# B&R Automation Studio project DuctLines (part 6)

#### Cyclic.ld
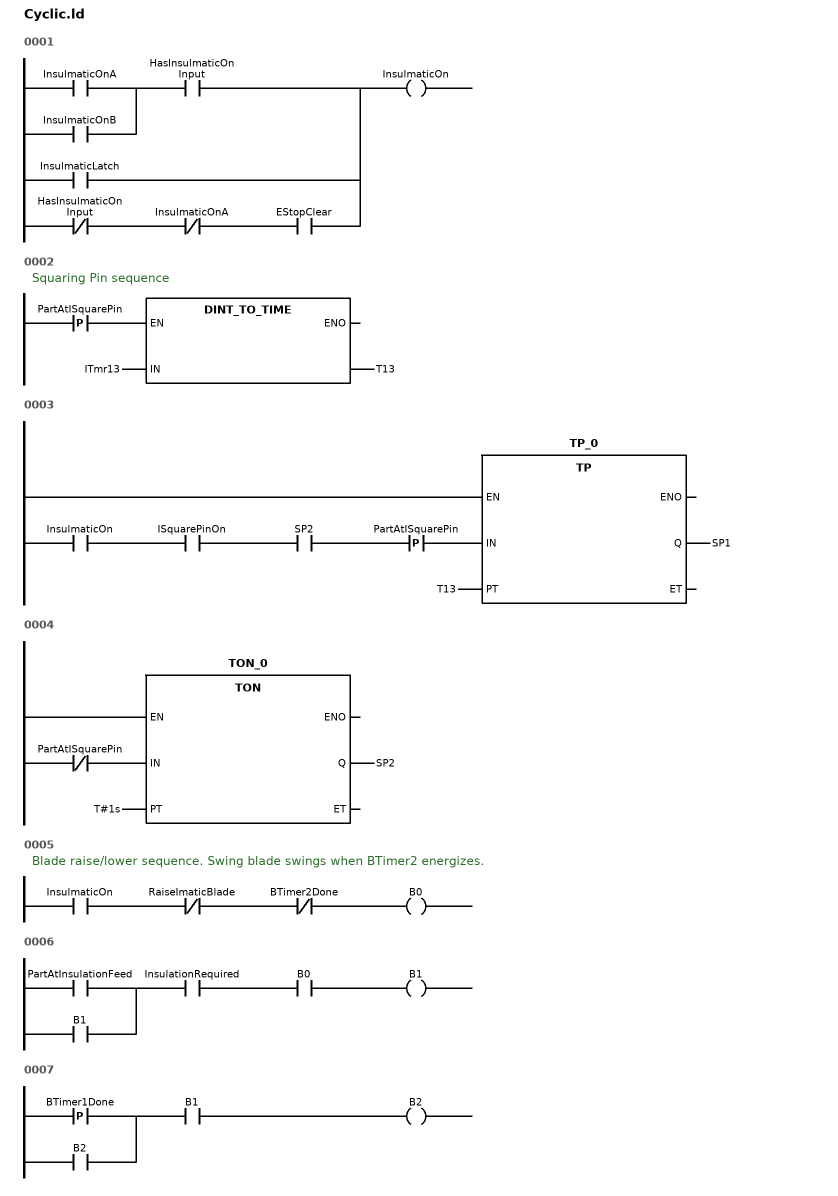
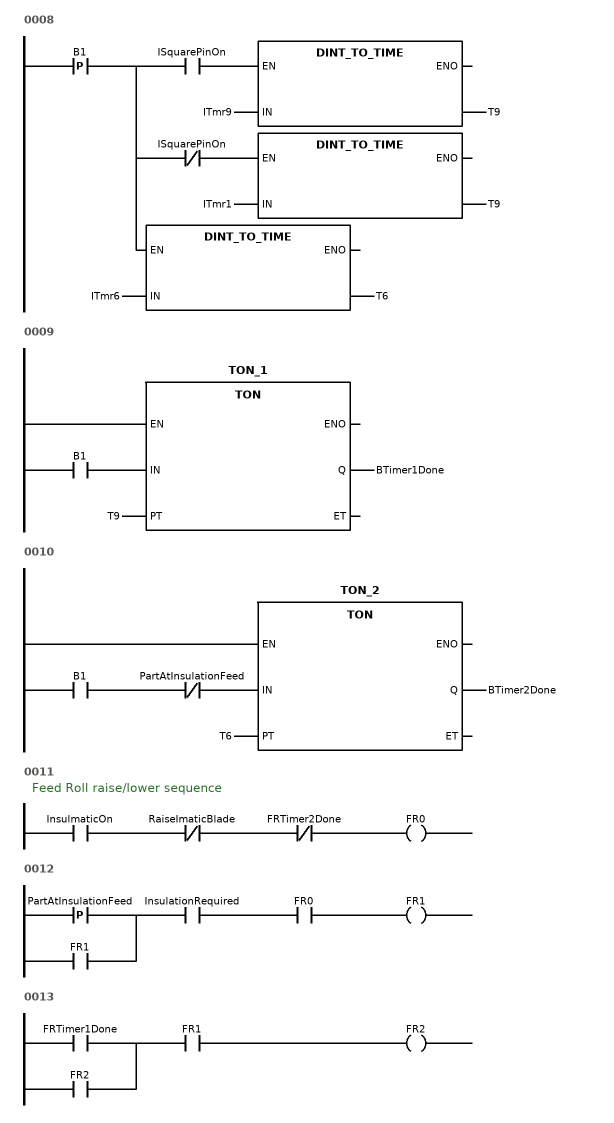
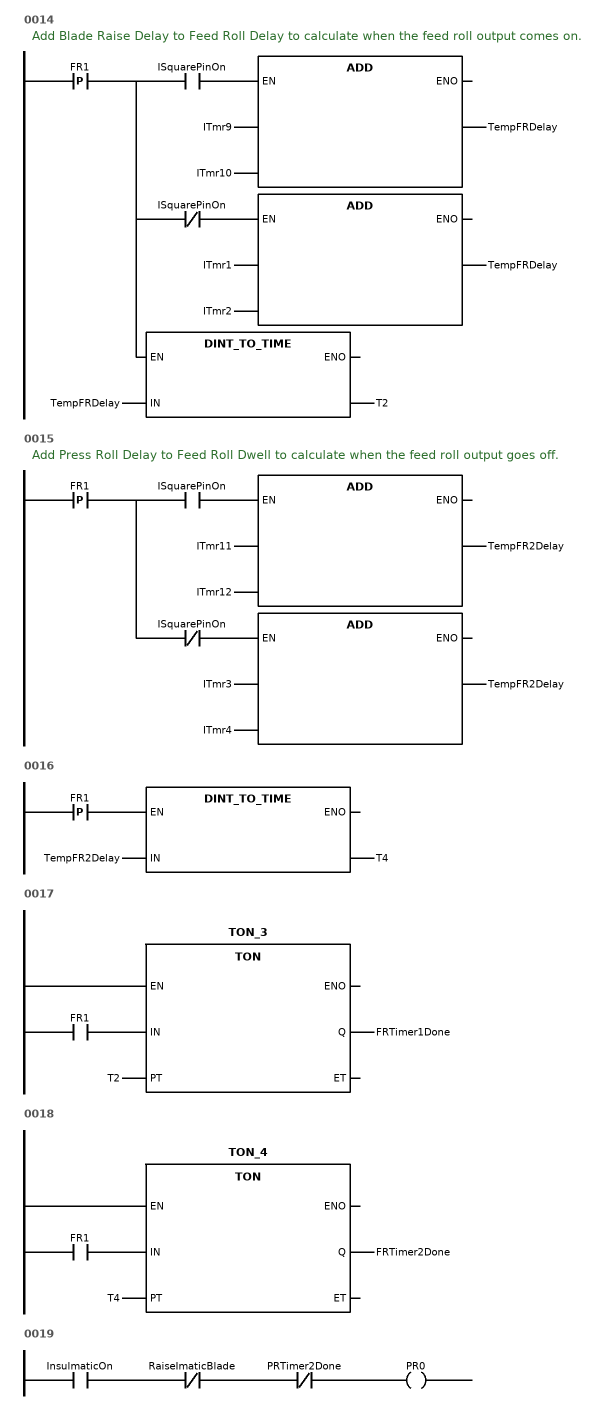
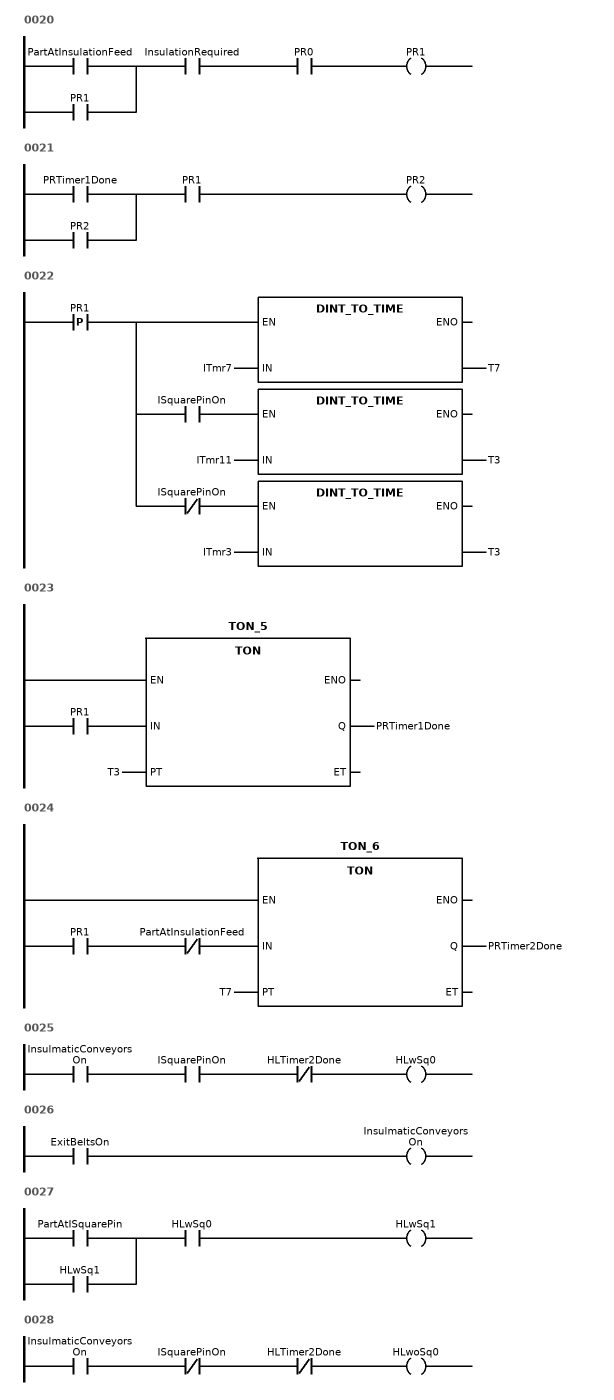
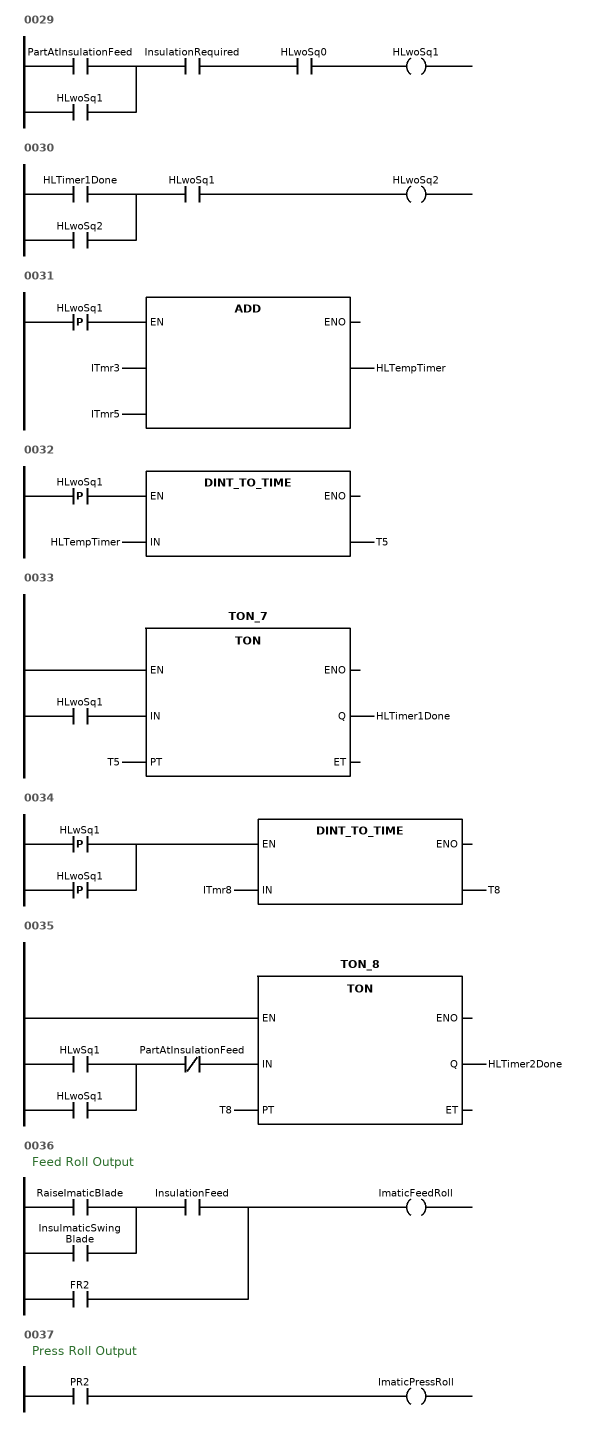
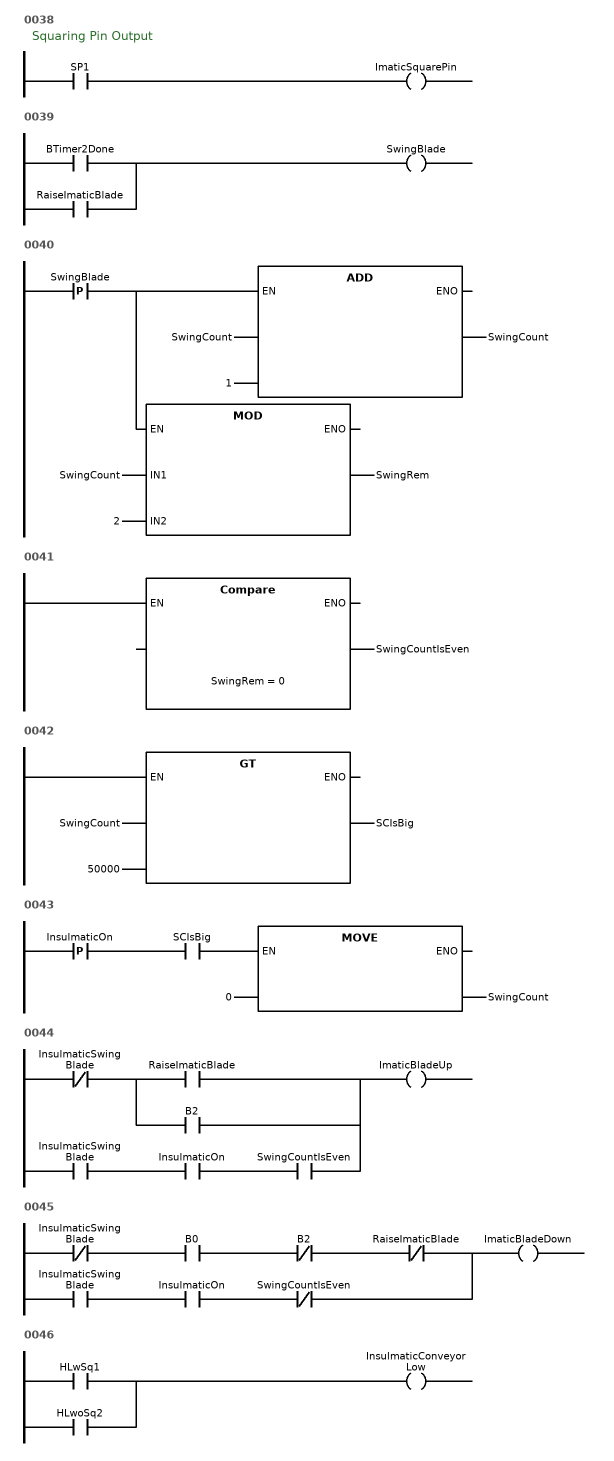
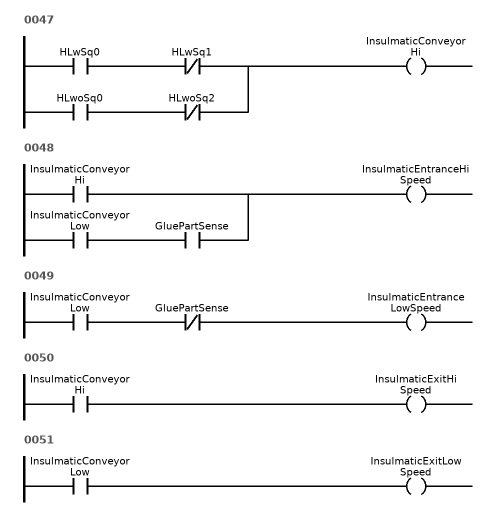
Ladder, written as Structured Text:
```iecst
PROGRAM _CYCLIC
VAR
    _e1 : R_TRIG;
    _e2 : R_TRIG;
    _e3 : R_TRIG;
    _e4 : R_TRIG;
    _e5 : R_TRIG;
    _e6 : R_TRIG;
    _e7 : R_TRIG;
    _e8 : R_TRIG;
    _e9 : R_TRIG;
    _e10 : R_TRIG;
    _e11 : R_TRIG;
    _e12 : R_TRIG;
    _e13 : R_TRIG;
    _e14 : R_TRIG;
    _e15 : R_TRIG;
END_VAR
(* Network 1 *)
InsulmaticOn := ((InsulmaticOnA OR InsulmaticOnB) AND HasInsulmaticOnInput) OR InsulmaticLatch OR (NOT HasInsulmaticOnInput AND NOT InsulmaticOnA AND EStopClear);

(* Network 2: Squaring Pin sequence *)
_e1(CLK := PartAtISquarePin);
IF _e1.Q THEN T13 := DINT_TO_TIME(ITmr13); END_IF;

(* Network 3 *)
_e2(CLK := PartAtISquarePin);
TP_0(IN := InsulmaticOn AND ISquarePinOn AND SP2 AND _e2.Q, PT := T13);
SP1 := TP_0.Q;

(* Network 4 *)
TON_0(IN := NOT PartAtISquarePin, PT := T#1s);
SP2 := TON_0.Q;

(* Network 5: Blade raise/lower sequence. Swing blade swings when BTimer2 energizes. *)
B0 := InsulmaticOn AND NOT RaiseImaticBlade AND NOT BTimer2Done;

(* Network 6 *)
B1 := (PartAtInsulationFeed OR B1) AND InsulationRequired AND B0;

(* Network 7 *)
_e3(CLK := BTimer1Done);
B2 := (_e3.Q OR B2) AND B1;

(* Network 8 *)
_e4(CLK := B1);
IF _e4.Q AND ISquarePinOn THEN T9 := DINT_TO_TIME(ITmr9); END_IF;
IF _e4.Q AND NOT ISquarePinOn THEN T9 := DINT_TO_TIME(ITmr1); END_IF;
IF _e4.Q THEN T6 := DINT_TO_TIME(ITmr6); END_IF;

(* Network 9 *)
TON_1(IN := B1, PT := T9);
BTimer1Done := TON_1.Q;

(* Network 10 *)
TON_2(IN := B1 AND NOT PartAtInsulationFeed, PT := T6);
BTimer2Done := TON_2.Q;

(* Network 11: Feed Roll raise/lower sequence *)
FR0 := InsulmaticOn AND NOT RaiseImaticBlade AND NOT FRTimer2Done;

(* Network 12 *)
_e5(CLK := PartAtInsulationFeed);
FR1 := (_e5.Q OR FR1) AND InsulationRequired AND FR0;

(* Network 13 *)
FR2 := (FRTimer1Done OR FR2) AND FR1;

(* Network 14: Add Blade Raise Delay to Feed Roll Delay to calculate when the feed roll output comes on. *)
_e6(CLK := FR1);
IF _e6.Q AND ISquarePinOn THEN TempFRDelay := ITmr9 + ITmr10; END_IF;
IF _e6.Q AND NOT ISquarePinOn THEN TempFRDelay := ITmr1 + ITmr2; END_IF;
IF _e6.Q THEN T2 := DINT_TO_TIME(TempFRDelay); END_IF;

(* Network 15: Add Press Roll Delay to Feed Roll Dwell to calculate when the feed roll output goes off. *)
_e7(CLK := FR1);
IF _e7.Q AND ISquarePinOn THEN TempFR2Delay := ITmr11 + ITmr12; END_IF;
IF _e7.Q AND NOT ISquarePinOn THEN TempFR2Delay := ITmr3 + ITmr4; END_IF;

(* Network 16 *)
_e8(CLK := FR1);
IF _e8.Q THEN T4 := DINT_TO_TIME(TempFR2Delay); END_IF;

(* Network 17 *)
TON_3(IN := FR1, PT := T2);
FRTimer1Done := TON_3.Q;

(* Network 18 *)
TON_4(IN := FR1, PT := T4);
FRTimer2Done := TON_4.Q;

(* Network 19 *)
PR0 := InsulmaticOn AND NOT RaiseImaticBlade AND NOT PRTimer2Done;

(* Network 20 *)
PR1 := (PartAtInsulationFeed OR PR1) AND InsulationRequired AND PR0;

(* Network 21 *)
PR2 := (PRTimer1Done OR PR2) AND PR1;

(* Network 22 *)
_e9(CLK := PR1);
IF _e9.Q THEN T7 := DINT_TO_TIME(ITmr7); END_IF;
IF _e9.Q AND ISquarePinOn THEN T3 := DINT_TO_TIME(ITmr11); END_IF;
IF _e9.Q AND NOT ISquarePinOn THEN T3 := DINT_TO_TIME(ITmr3); END_IF;

(* Network 23 *)
TON_5(IN := PR1, PT := T3);
PRTimer1Done := TON_5.Q;

(* Network 24 *)
TON_6(IN := PR1 AND NOT PartAtInsulationFeed, PT := T7);
PRTimer2Done := TON_6.Q;

(* Network 25 *)
HLwSq0 := InsulmaticConveyorsOn AND ISquarePinOn AND NOT HLTimer2Done;

(* Network 26 *)
InsulmaticConveyorsOn := ExitBeltsOn;

(* Network 27 *)
HLwSq1 := (PartAtISquarePin OR HLwSq1) AND HLwSq0;

(* Network 28 *)
HLwoSq0 := InsulmaticConveyorsOn AND NOT ISquarePinOn AND NOT HLTimer2Done;

(* Network 29 *)
HLwoSq1 := (PartAtInsulationFeed OR HLwoSq1) AND InsulationRequired AND HLwoSq0;

(* Network 30 *)
HLwoSq2 := (HLTimer1Done OR HLwoSq2) AND HLwoSq1;

(* Network 31 *)
_e10(CLK := HLwoSq1);
IF _e10.Q THEN HLTempTimer := ITmr3 + ITmr5; END_IF;

(* Network 32 *)
_e11(CLK := HLwoSq1);
IF _e11.Q THEN T5 := DINT_TO_TIME(HLTempTimer); END_IF;

(* Network 33 *)
TON_7(IN := HLwoSq1, PT := T5);
HLTimer1Done := TON_7.Q;

(* Network 34 *)
_e12(CLK := HLwSq1);
_e13(CLK := HLwoSq1);
IF _e12.Q OR _e13.Q THEN T8 := DINT_TO_TIME(ITmr8); END_IF;

(* Network 35 *)
TON_8(IN := (HLwSq1 OR HLwoSq1) AND NOT PartAtInsulationFeed, PT := T8);
HLTimer2Done := TON_8.Q;

(* Network 36: Feed Roll Output *)
ImaticFeedRoll := ((RaiseImaticBlade OR InsulmaticSwingBlade) AND InsulationFeed) OR FR2;

(* Network 37: Press Roll Output *)
ImaticPressRoll := PR2;

(* Network 38: Squaring Pin Output *)
ImaticSquarePin := SP1;

(* Network 39 *)
SwingBlade := BTimer2Done OR RaiseImaticBlade;

(* Network 40 *)
_e14(CLK := SwingBlade);
IF _e14.Q THEN
    SwingCount := SwingCount + 1;
    SwingRem := SwingCount MOD 2;
END_IF;

(* Network 41 *)
SwingCountIsEven := SwingRem = 0;

(* Network 42 *)
SCIsBig := SwingCount > 50000;

(* Network 43 *)
_e15(CLK := InsulmaticOn);
IF _e15.Q AND SCIsBig THEN SwingCount := 0; END_IF;

(* Network 44 *)
ImaticBladeUp := (NOT InsulmaticSwingBlade AND (RaiseImaticBlade OR B2)) OR (InsulmaticSwingBlade AND InsulmaticOn AND SwingCountIsEven);

(* Network 45 *)
ImaticBladeDown := (NOT InsulmaticSwingBlade AND B0 AND NOT B2 AND NOT RaiseImaticBlade) OR (InsulmaticSwingBlade AND InsulmaticOn AND NOT SwingCountIsEven);

(* Network 46 *)
InsulmaticConveyorLow := HLwSq1 OR HLwoSq2;

(* Network 47 *)
InsulmaticConveyorHi := (HLwSq0 AND NOT HLwSq1) OR (HLwoSq0 AND NOT HLwoSq2);

(* Network 48 *)
InsulmaticEntranceHiSpeed := InsulmaticConveyorHi OR (InsulmaticConveyorLow AND GluePartSense);

(* Network 49 *)
InsulmaticEntranceLowSpeed := InsulmaticConveyorLow AND NOT GluePartSense;

(* Network 50 *)
InsulmaticExitHiSpeed := InsulmaticConveyorHi;

(* Network 51 *)
InsulmaticExitLowSpeed := InsulmaticConveyorLow;
END_PROGRAM
```

### Program Logical/Pinspotter (IEC)

#### Variables.var
```iecst
VAR
	PS0 : BOOL;
	EncoderReset : BOOL;
	PS1 : BOOL;
	PinSpaceSelector : USINT;
	RepeatCounter : DINT;
	Target : DINT;
	PinSpacing : REAL;
	PinSpaceSelectorIs9 : BOOL;
	RealTarget : REAL;
	RealCounts : REAL;
	Drive : BOOL;
	DriveComplete : BOOL;
	DriveDwell : TIME;
	PS3 : BOOL;
	PS2 : BOOL;
	UpDateSignal : BOOL;
	IndexFinished : BOOL;
	PinningDone : BOOL;
	PS4 : BOOL;
	PinAgain : BOOL;
	TON_2 : TON;
	DelayTime : TIME;
	TP_1 : TP;
	LoadDelayPulse : BOOL;
	PinLoadTime : TIME;
	TP_2 : TP;
	TON_0 : TON;
	RCounterIs0 : BOOL;
END_VAR
```

#### Cyclic.ld
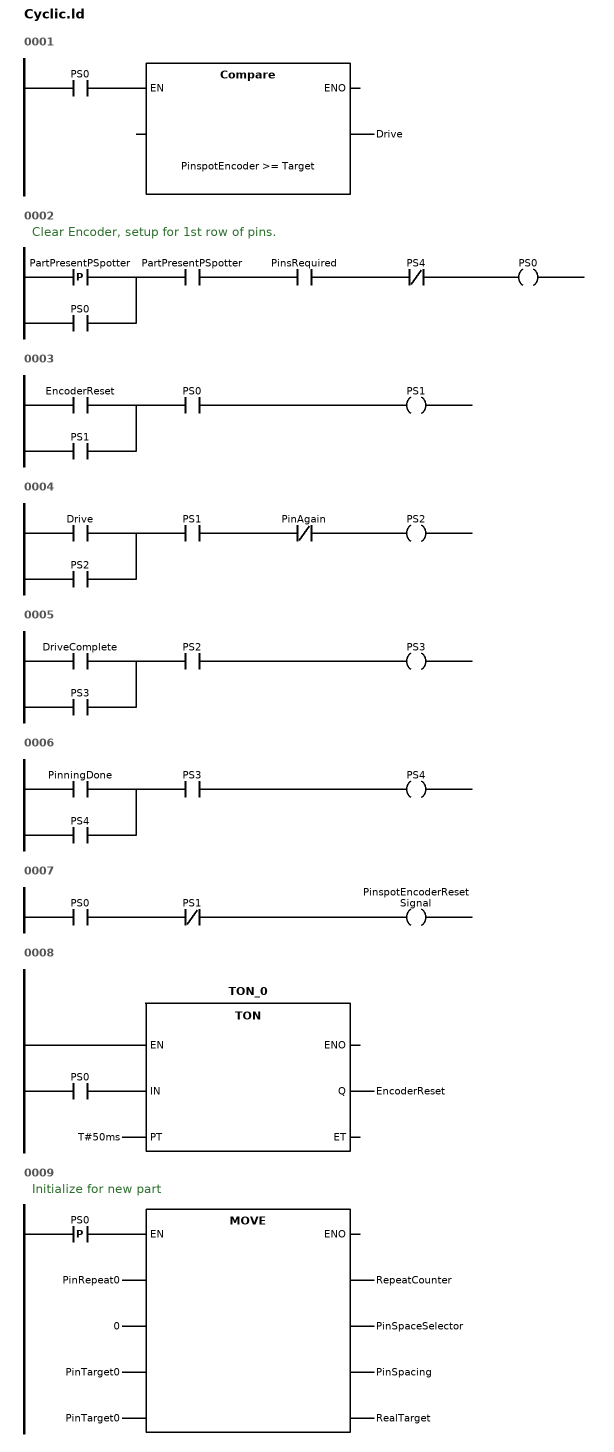
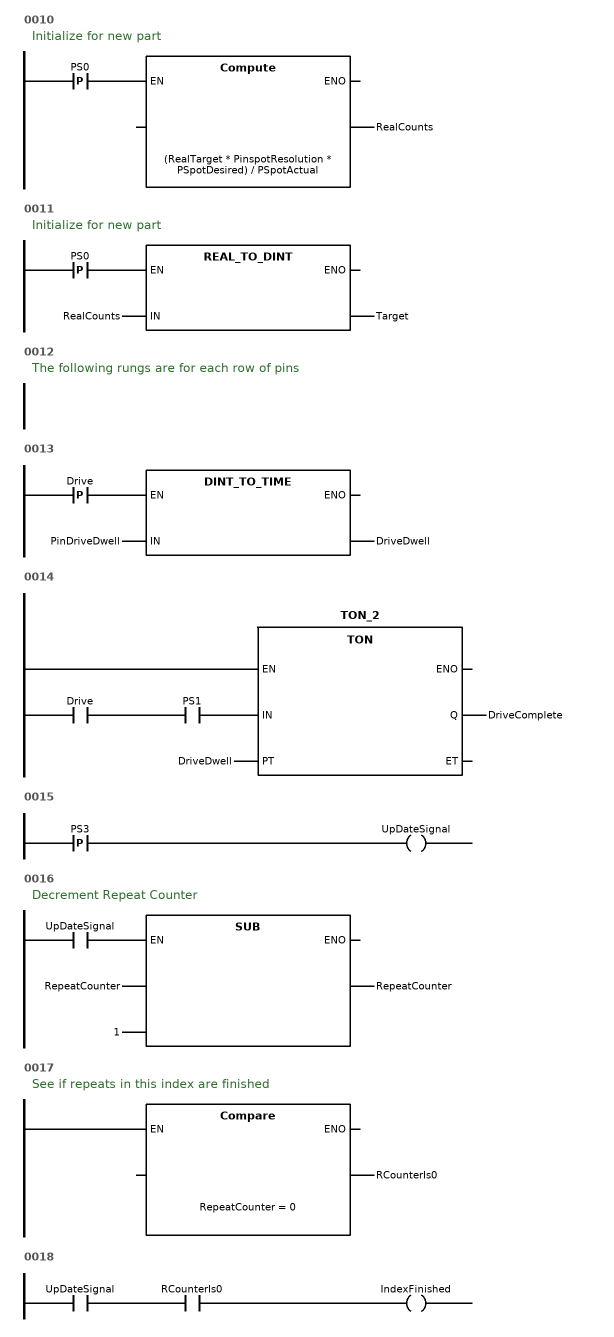
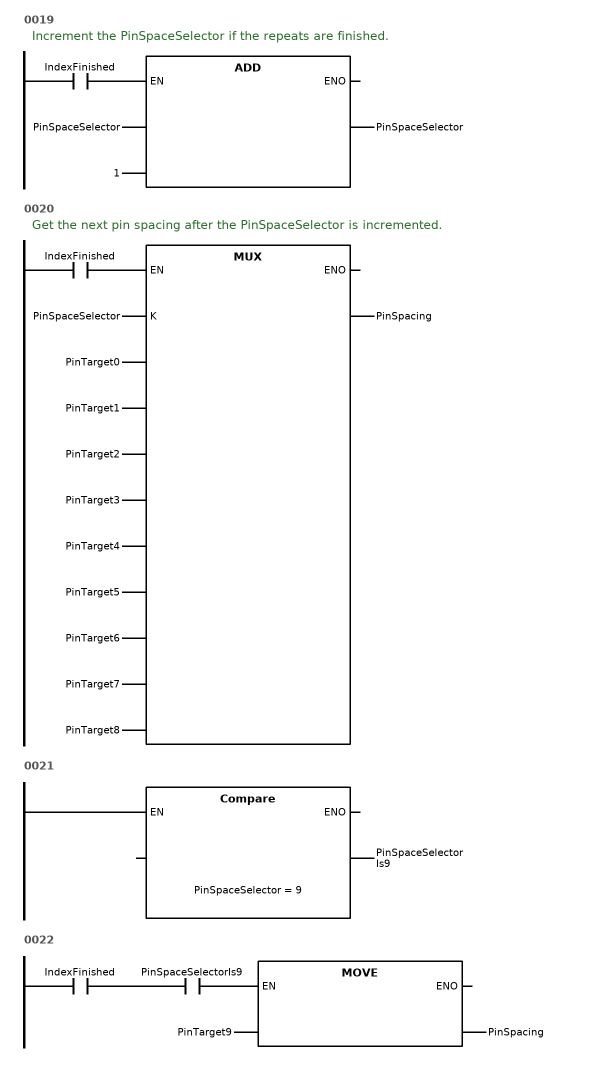
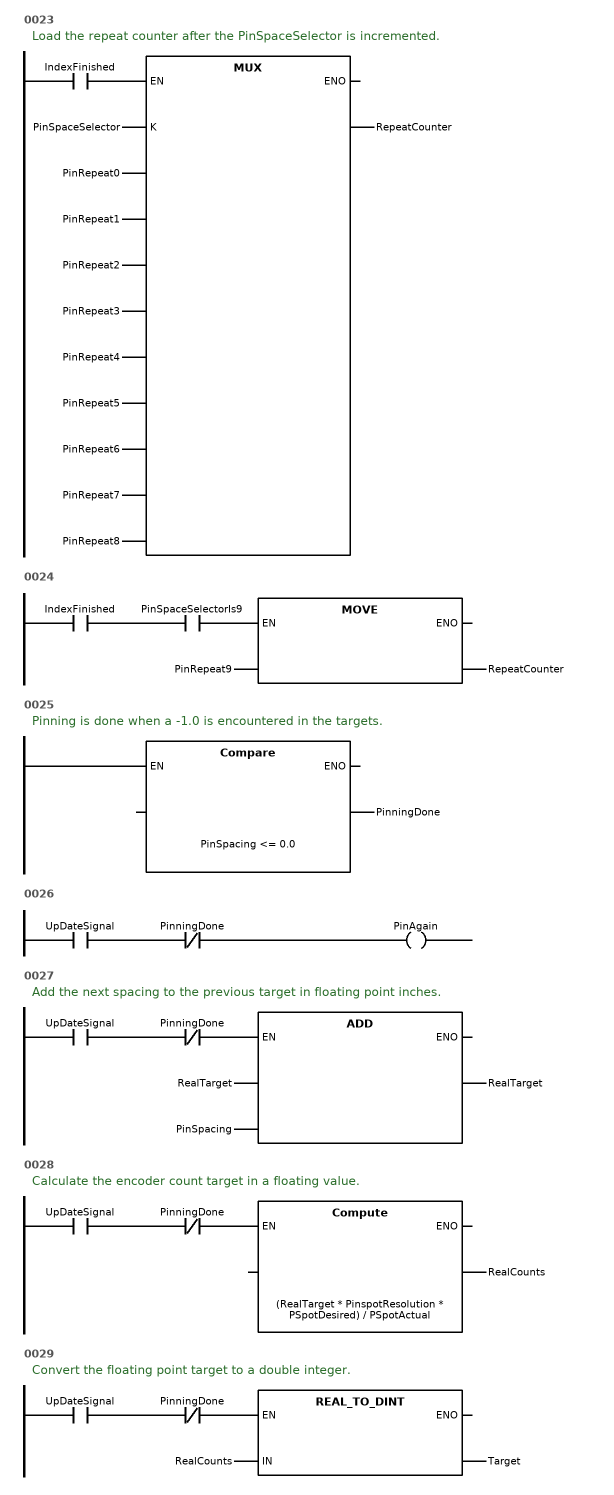
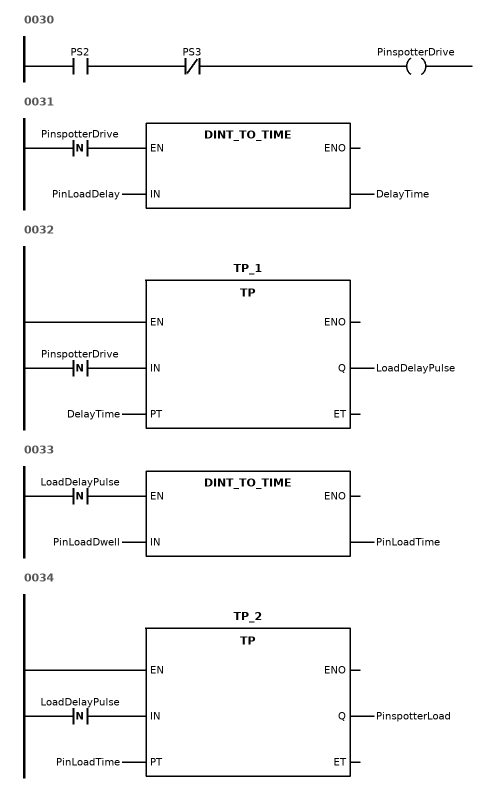
Ladder, written as Structured Text:
```iecst
PROGRAM _CYCLIC
VAR
    _e1 : R_TRIG;
    _e2 : R_TRIG;
    _e3 : R_TRIG;
    _e4 : R_TRIG;
    _e5 : R_TRIG;
    _e6 : R_TRIG;
    _e7 : F_TRIG;
    _e8 : F_TRIG;
    _e9 : F_TRIG;
    _e10 : F_TRIG;
END_VAR
(* Network 1 *)
IF PS0 THEN Drive := PinspotEncoder >= Target; END_IF;

(* Network 2: Clear Encoder, setup for 1st row of pins. *)
_e1(CLK := PartPresentPSpotter);
PS0 := (_e1.Q OR PS0) AND PartPresentPSpotter AND PinsRequired AND NOT PS4;

(* Network 3 *)
PS1 := (EncoderReset OR PS1) AND PS0;

(* Network 4 *)
PS2 := (Drive OR PS2) AND PS1 AND NOT PinAgain;

(* Network 5 *)
PS3 := (DriveComplete OR PS3) AND PS2;

(* Network 6 *)
PS4 := (PinningDone OR PS4) AND PS3;

(* Network 7 *)
PinspotEncoderResetSignal := PS0 AND NOT PS1;

(* Network 8 *)
TON_0(IN := PS0, PT := T#50ms);
EncoderReset := TON_0.Q;

(* Network 9: Initialize for new part *)
_e2(CLK := PS0);
IF _e2.Q THEN
    RepeatCounter := PinRepeat0;
    PinSpaceSelector := 0;
    PinSpacing := PinTarget0;
    RealTarget := PinTarget0;
END_IF;

(* Network 10: Initialize for new part *)
_e3(CLK := PS0);
IF _e3.Q THEN RealCounts := (RealTarget * PinspotResolution * PSpotDesired) / PSpotActual; END_IF;

(* Network 11: Initialize for new part *)
_e4(CLK := PS0);
IF _e4.Q THEN Target := REAL_TO_DINT(RealCounts); END_IF;

(* Network 12: The following rungs are for each row of pins *)

(* Network 13 *)
_e5(CLK := Drive);
IF _e5.Q THEN DriveDwell := DINT_TO_TIME(PinDriveDwell); END_IF;

(* Network 14 *)
TON_2(IN := Drive AND PS1, PT := DriveDwell);
DriveComplete := TON_2.Q;

(* Network 15 *)
_e6(CLK := PS3);
UpDateSignal := _e6.Q;

(* Network 16: Decrement Repeat Counter *)
IF UpDateSignal THEN RepeatCounter := RepeatCounter - 1; END_IF;

(* Network 17: See if repeats in this index are finished *)
RCounterIs0 := RepeatCounter = 0;

(* Network 18 *)
IndexFinished := UpDateSignal AND RCounterIs0;

(* Network 19: Increment the PinSpaceSelector if the repeats are finished. *)
IF IndexFinished THEN PinSpaceSelector := PinSpaceSelector + 1; END_IF;

(* Network 20: Get the next pin spacing after the PinSpaceSelector is incremented. *)
IF IndexFinished THEN
    PinSpacing := MUX(K := PinSpaceSelector, IN2 := PinTarget0, IN3 := PinTarget1, IN4 := PinTarget2, IN5 := PinTarget3, IN6 := PinTarget4, IN7 := PinTarget5, IN8 := PinTarget6, IN9 := PinTarget7, IN10 := PinTarget8);
END_IF;

(* Network 21 *)
PinSpaceSelectorIs9 := PinSpaceSelector = 9;

(* Network 22 *)
IF IndexFinished AND PinSpaceSelectorIs9 THEN PinSpacing := PinTarget9; END_IF;

(* Network 23: Load the repeat counter after the PinSpaceSelector is incremented. *)
IF IndexFinished THEN
    RepeatCounter := MUX(K := PinSpaceSelector, IN2 := PinRepeat0, IN3 := PinRepeat1, IN4 := PinRepeat2, IN5 := PinRepeat3, IN6 := PinRepeat4, IN7 := PinRepeat5, IN8 := PinRepeat6, IN9 := PinRepeat7, IN10 := PinRepeat8);
END_IF;

(* Network 24 *)
IF IndexFinished AND PinSpaceSelectorIs9 THEN RepeatCounter := PinRepeat9; END_IF;

(* Network 25: Pinning is done when a -1.0 is encountered in the targets. *)
PinningDone := PinSpacing <= 0.0;

(* Network 26 *)
PinAgain := UpDateSignal AND NOT PinningDone;

(* Network 27: Add the next spacing to the previous target in floating point inches. *)
IF UpDateSignal AND NOT PinningDone THEN RealTarget := RealTarget + PinSpacing; END_IF;

(* Network 28: Calculate the encoder count target in a floating value.  *)
IF UpDateSignal AND NOT PinningDone THEN
    RealCounts := (RealTarget * PinspotResolution * PSpotDesired) / PSpotActual;
END_IF;

(* Network 29: Convert the floating point target to a double integer. *)
IF UpDateSignal AND NOT PinningDone THEN Target := REAL_TO_DINT(RealCounts); END_IF;

(* Network 30 *)
PinspotterDrive := PS2 AND NOT PS3;

(* Network 31 *)
_e7(CLK := PinspotterDrive);
IF _e7.Q THEN DelayTime := DINT_TO_TIME(PinLoadDelay); END_IF;

(* Network 32 *)
_e8(CLK := PinspotterDrive);
TP_1(IN := _e8.Q, PT := DelayTime);
LoadDelayPulse := TP_1.Q;

(* Network 33 *)
_e9(CLK := LoadDelayPulse);
IF _e9.Q THEN PinLoadTime := DINT_TO_TIME(PinLoadDwell); END_IF;

(* Network 34 *)
_e10(CLK := LoadDelayPulse);
TP_2(IN := _e10.Q, PT := PinLoadTime);
PinspotterLoad := TP_2.Q;
END_PROGRAM
```

### Program Logical/BrakeCommon (IEC) - In this file: The encoder feedback is scaled to inches. All of the brakes use real dimensions, except for the Electric Servo Brake, The Auto Latch for all brake styles, Target selection for all brake styles, A latch that holds all outputs in their initial state, The bending routine for all brakes without their own PLC begins about rung 29, Clamp, Leaf, Beam outputs for brakes without a PLC begins about rung 42, Brake Conveyor and Auto/Man Indicator Outputs

#### Variables.var
```iecst
VAR
	BAOK : BOOL;
	BCTGreatThan0 : BOOL;
	BDOK : BOOL;
	BeamSettleTimerDone : BOOL;
	BrakeSetOK : BOOL;
	EWBAutoLatch : BOOL;
	JobsDifferent : BOOL;
	MakeTargets : BOOL;
	RaiseLeafTimerDone : BOOL;
	RawBrakeEncoder : REAL;
	RefSignalReset : BOOL;
	ResOK : BOOL;
	SetSignalReset : BOOL;
	SingleCyclingBrake : BOOL;
	StopLeafTimerDone : BOOL;
	TON_0 : TON;
	TON_1 : TON;
	TON_2 : TON;
	TON_3 : TON;
	TON_4 : TON;
	WBBeamSettleStep : BOOL;
	WBCheckBeamStep : BOOL;
	WBCheckLeafStep : BOOL;
	WBIndex : INT;
	WBLeafNotHomeStep : BOOL;
	WBLowerBeamStep : BOOL;
	WBLowerLeafStep : BOOL;
	WBRaiseBeamStep : BOOL;
	WBStopLeafStep : BOOL;
END_VAR
```

#### Cyclic.ld
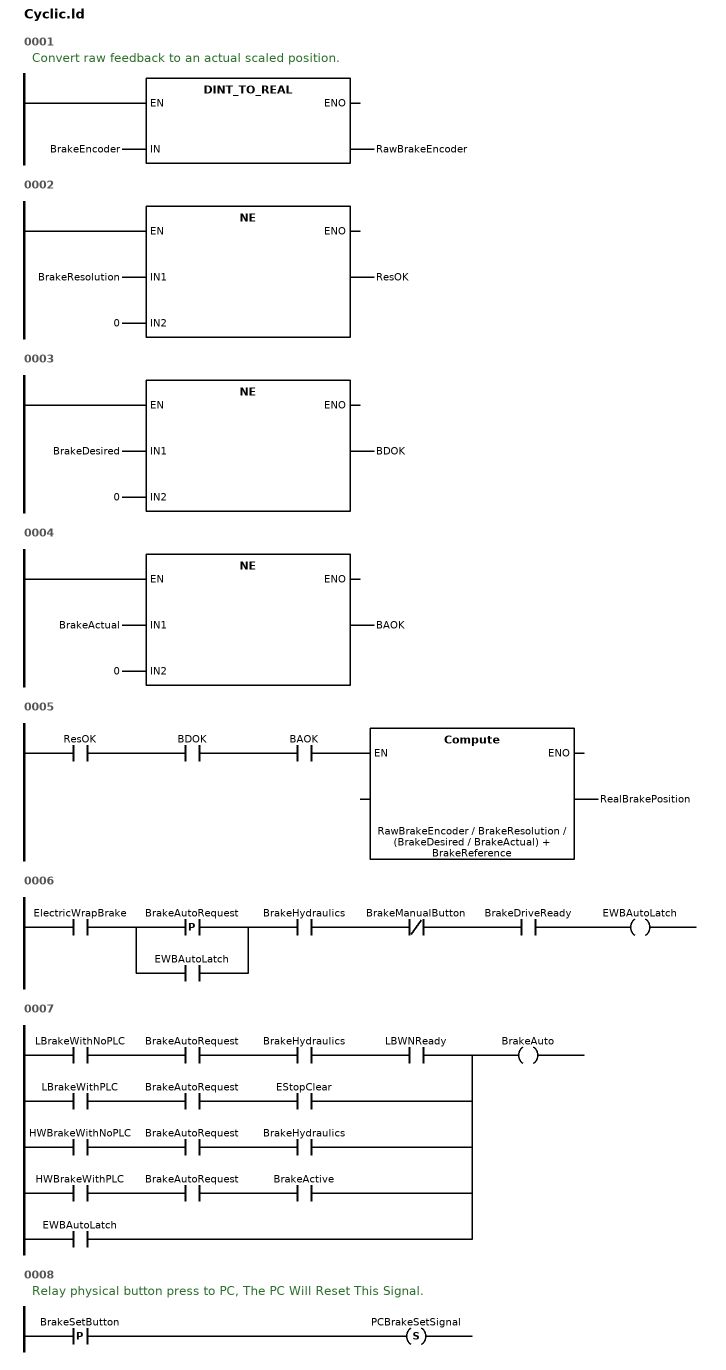
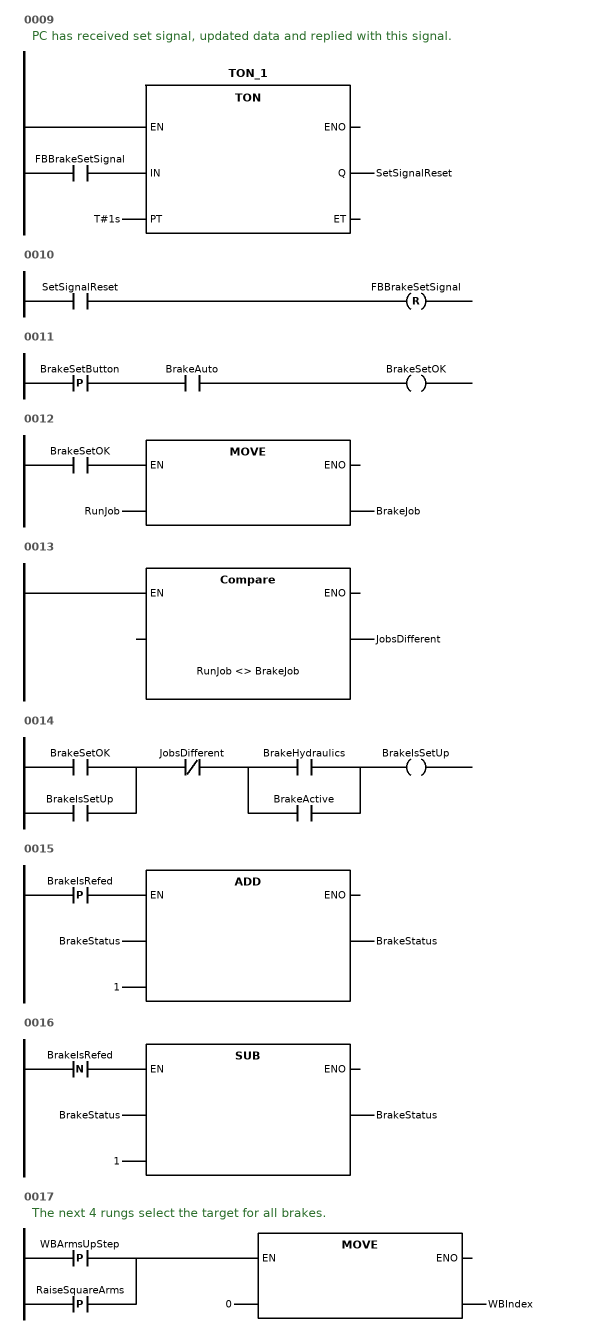
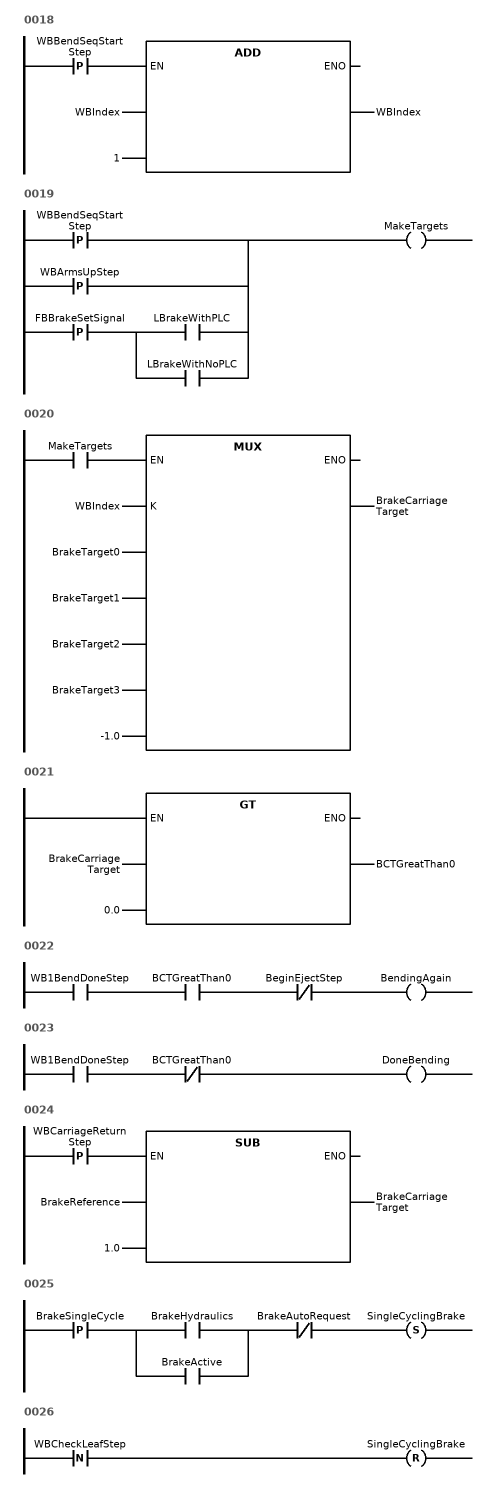
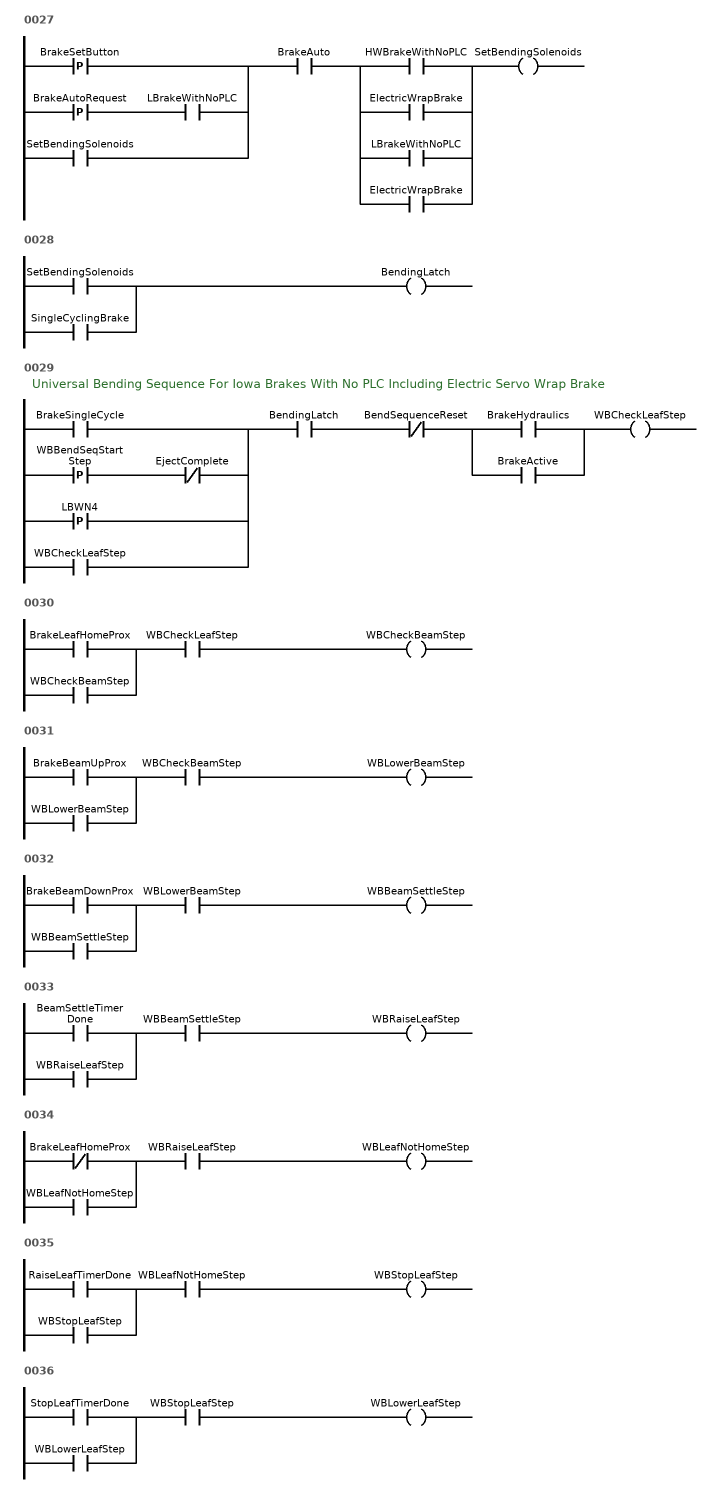
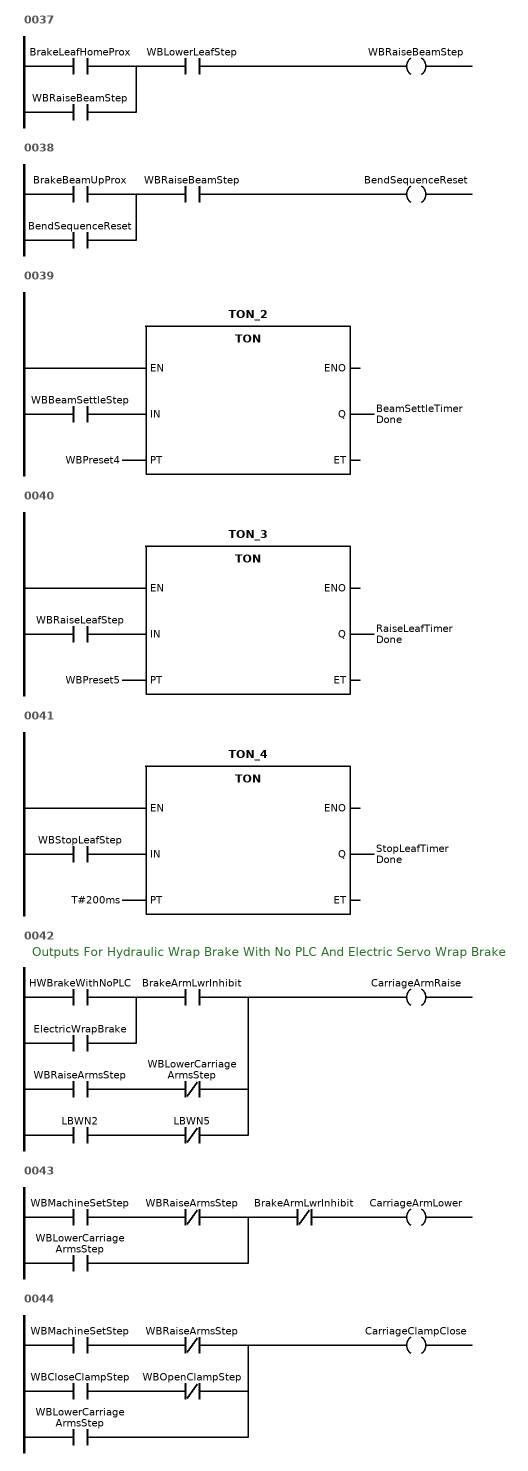
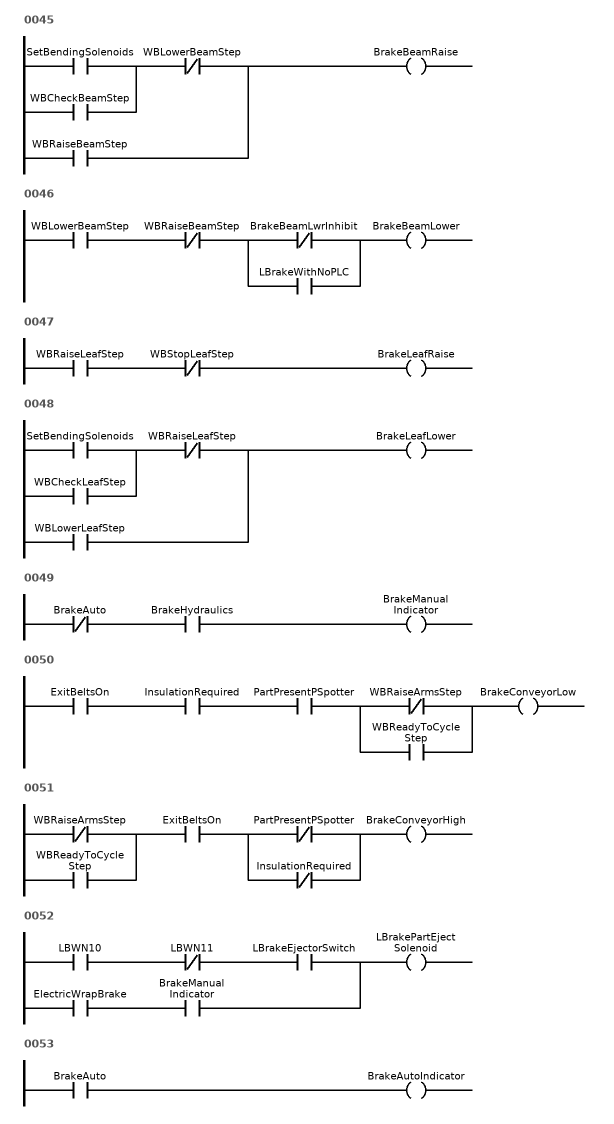
Ladder, written as Structured Text:
```iecst
PROGRAM _CYCLIC
VAR
    _e1 : R_TRIG;
    _e2 : R_TRIG;
    _e3 : R_TRIG;
    _p4 : BOOL;
    _e5 : R_TRIG;
    _e6 : F_TRIG;
    _e7 : R_TRIG;
    _e8 : R_TRIG;
    _e9 : R_TRIG;
    _e10 : R_TRIG;
    _e11 : R_TRIG;
    _e12 : R_TRIG;
    _e13 : R_TRIG;
    _e14 : R_TRIG;
    _e15 : F_TRIG;
    _e16 : R_TRIG;
    _e17 : R_TRIG;
    _p18 : BOOL;
    _e19 : R_TRIG;
    _e20 : R_TRIG;
    _p21 : BOOL;
    _p22 : BOOL;
    _p23 : BOOL;
END_VAR
(* Network 1: Convert raw feedback to an actual scaled position. *)
RawBrakeEncoder := DINT_TO_REAL(BrakeEncoder);

(* Network 2 *)
ResOK := BrakeResolution <> 0;

(* Network 3 *)
BDOK := BrakeDesired <> 0;

(* Network 4 *)
BAOK := BrakeActual <> 0;

(* Network 5 *)
IF ResOK AND BDOK AND BAOK THEN
    RealBrakePosition := RawBrakeEncoder / BrakeResolution / (BrakeDesired / BrakeActual) + BrakeReference;
END_IF;

(* Network 6 *)
_e1(CLK := BrakeAutoRequest);
EWBAutoLatch := ElectricWrapBrake AND (_e1.Q OR EWBAutoLatch) AND BrakeHydraulics AND NOT BrakeManualButton AND BrakeDriveReady;

(* Network 7 *)
BrakeAuto := (LBrakeWithNoPLC AND BrakeAutoRequest AND BrakeHydraulics AND LBWNReady) OR (LBrakeWithPLC AND BrakeAutoRequest AND EStopClear) OR (HWBrakeWithNoPLC AND BrakeAutoRequest AND BrakeHydraulics) OR (HWBrakeWithPLC AND BrakeAutoRequest AND BrakeActive) OR EWBAutoLatch;

(* Network 8: Relay physical button press to PC, The PC Will Reset This Signal. *)
_e2(CLK := BrakeSetButton);
IF _e2.Q THEN PCBrakeSetSignal := TRUE; END_IF;

(* Network 9: PC has received set signal, updated data and replied with this signal. *)
TON_1(IN := FBBrakeSetSignal, PT := T#1s);
SetSignalReset := TON_1.Q;

(* Network 10 *)
IF SetSignalReset THEN FBBrakeSetSignal := FALSE; END_IF;

(* Network 11 *)
_e3(CLK := BrakeSetButton);
BrakeSetOK := _e3.Q AND BrakeAuto;

(* Network 12 *)
IF BrakeSetOK THEN BrakeJob := RunJob; END_IF;

(* Network 13 *)
JobsDifferent := RunJob <> BrakeJob;

(* Network 14 *)
_p4 := (BrakeSetOK OR BrakeIsSetUp) AND NOT JobsDifferent;
BrakeIsSetUp := _p4 AND (BrakeHydraulics OR BrakeActive);

(* Network 15 *)
_e5(CLK := BrakeIsRefed);
IF _e5.Q THEN BrakeStatus := BrakeStatus + 1; END_IF;

(* Network 16 *)
_e6(CLK := BrakeIsRefed);
IF _e6.Q THEN BrakeStatus := BrakeStatus - 1; END_IF;

(* Network 17: The next 4 rungs select the target for all brakes. *)
_e7(CLK := WBArmsUpStep);
_e8(CLK := RaiseSquareArms);
IF _e7.Q OR _e8.Q THEN WBIndex := 0; END_IF;

(* Network 18 *)
_e9(CLK := WBBendSeqStartStep);
IF _e9.Q THEN WBIndex := WBIndex + 1; END_IF;

(* Network 19 *)
_e10(CLK := WBBendSeqStartStep);
_e11(CLK := WBArmsUpStep);
_e12(CLK := FBBrakeSetSignal);
MakeTargets := _e10.Q OR _e11.Q OR (_e12.Q AND (LBrakeWithPLC OR LBrakeWithNoPLC));

(* Network 20 *)
IF MakeTargets THEN
    BrakeCarriageTarget := MUX(K := WBIndex, IN2 := BrakeTarget0, IN3 := BrakeTarget1, IN4 := BrakeTarget2, IN5 := BrakeTarget3, IN6 := -1.0);
END_IF;

(* Network 21 *)
BCTGreatThan0 := BrakeCarriageTarget > 0.0;

(* Network 22 *)
BendingAgain := WB1BendDoneStep AND BCTGreatThan0 AND NOT BeginEjectStep;

(* Network 23 *)
DoneBending := WB1BendDoneStep AND NOT BCTGreatThan0;

(* Network 24 *)
_e13(CLK := WBCarriageReturnStep);
IF _e13.Q THEN BrakeCarriageTarget := BrakeReference - 1.0; END_IF;

(* Network 25 *)
_e14(CLK := BrakeSingleCycle);
IF _e14.Q AND (BrakeHydraulics OR BrakeActive) AND NOT BrakeAutoRequest THEN
    SingleCyclingBrake := TRUE;
END_IF;

(* Network 26 *)
_e15(CLK := WBCheckLeafStep);
IF _e15.Q THEN SingleCyclingBrake := FALSE; END_IF;

(* Network 27 *)
_e16(CLK := BrakeSetButton);
_e17(CLK := BrakeAutoRequest);
_p18 := (_e16.Q OR (_e17.Q AND LBrakeWithNoPLC) OR SetBendingSolenoids) AND BrakeAuto;
SetBendingSolenoids := _p18 AND (HWBrakeWithNoPLC OR ElectricWrapBrake OR LBrakeWithNoPLC);

(* Network 28 *)
BendingLatch := SetBendingSolenoids OR SingleCyclingBrake;

(* Network 29: Universal Bending Sequence For Iowa Brakes With No PLC Including Electric Servo Wrap Brake *)
_e19(CLK := WBBendSeqStartStep);
_e20(CLK := LBWN4);
_p21 := (BrakeSingleCycle OR (_e19.Q AND NOT EjectComplete) OR _e20.Q OR WBCheckLeafStep) AND BendingLatch AND NOT BendSequenceReset;
WBCheckLeafStep := _p21 AND (BrakeHydraulics OR BrakeActive);

(* Network 30 *)
WBCheckBeamStep := (BrakeLeafHomeProx OR WBCheckBeamStep) AND WBCheckLeafStep;

(* Network 31 *)
WBLowerBeamStep := (BrakeBeamUpProx OR WBLowerBeamStep) AND WBCheckBeamStep;

(* Network 32 *)
WBBeamSettleStep := (BrakeBeamDownProx OR WBBeamSettleStep) AND WBLowerBeamStep;

(* Network 33 *)
WBRaiseLeafStep := (BeamSettleTimerDone OR WBRaiseLeafStep) AND WBBeamSettleStep;

(* Network 34 *)
WBLeafNotHomeStep := (NOT BrakeLeafHomeProx OR WBLeafNotHomeStep) AND WBRaiseLeafStep;

(* Network 35 *)
WBStopLeafStep := (RaiseLeafTimerDone OR WBStopLeafStep) AND WBLeafNotHomeStep;

(* Network 36 *)
WBLowerLeafStep := (StopLeafTimerDone OR WBLowerLeafStep) AND WBStopLeafStep;

(* Network 37 *)
WBRaiseBeamStep := (BrakeLeafHomeProx OR WBRaiseBeamStep) AND WBLowerLeafStep;

(* Network 38 *)
BendSequenceReset := (BrakeBeamUpProx OR BendSequenceReset) AND WBRaiseBeamStep;

(* Network 39 *)
TON_2(IN := WBBeamSettleStep, PT := WBPreset4);
BeamSettleTimerDone := TON_2.Q;

(* Network 40 *)
TON_3(IN := WBRaiseLeafStep, PT := WBPreset5);
RaiseLeafTimerDone := TON_3.Q;

(* Network 41 *)
TON_4(IN := WBStopLeafStep, PT := T#200ms);
StopLeafTimerDone := TON_4.Q;

(* Network 42: Outputs For Hydraulic Wrap Brake With No PLC And Electric Servo Wrap Brake *)
CarriageArmRaise := ((HWBrakeWithNoPLC OR ElectricWrapBrake) AND BrakeArmLwrInhibit) OR (WBRaiseArmsStep AND NOT WBLowerCarriageArmsStep) OR (LBWN2 AND NOT LBWN5);

(* Network 43 *)
CarriageArmLower := ((WBMachineSetStep AND NOT WBRaiseArmsStep) OR WBLowerCarriageArmsStep) AND NOT BrakeArmLwrInhibit;

(* Network 44 *)
CarriageClampClose := (WBMachineSetStep AND NOT WBRaiseArmsStep) OR (WBCloseClampStep AND NOT WBOpenClampStep) OR WBLowerCarriageArmsStep;

(* Network 45 *)
BrakeBeamRaise := ((SetBendingSolenoids OR WBCheckBeamStep) AND NOT WBLowerBeamStep) OR WBRaiseBeamStep;

(* Network 46 *)
BrakeBeamLower := WBLowerBeamStep AND NOT WBRaiseBeamStep AND (NOT BrakeBeamLwrInhibit OR LBrakeWithNoPLC);

(* Network 47 *)
BrakeLeafRaise := WBRaiseLeafStep AND NOT WBStopLeafStep;

(* Network 48 *)
BrakeLeafLower := ((SetBendingSolenoids OR WBCheckLeafStep) AND NOT WBRaiseLeafStep) OR WBLowerLeafStep;

(* Network 49 *)
BrakeManualIndicator := NOT BrakeAuto AND BrakeHydraulics;

(* Network 50 *)
_p22 := ExitBeltsOn AND InsulationRequired AND PartPresentPSpotter;
BrakeConveyorLow := _p22 AND (NOT WBRaiseArmsStep OR WBReadyToCycleStep);

(* Network 51 *)
_p23 := (NOT WBRaiseArmsStep OR WBReadyToCycleStep) AND ExitBeltsOn;
BrakeConveyorHigh := _p23 AND (NOT PartPresentPSpotter OR NOT InsulationRequired);

(* Network 52 *)
LBrakePartEjectSolenoid := (LBWN10 AND NOT LBWN11 AND LBrakeEjectorSwitch) OR (ElectricWrapBrake AND BrakeManualIndicator);

(* Network 53 *)
BrakeAutoIndicator := BrakeAuto;
END_PROGRAM
```

### Program Logical/HWBwoPLC (IEC)

#### Variables.var
```iecst
VAR
	EjectTimerDone : BOOL;
	PositionGreaterThan12 : BOOL;
	PPDTimerDone : BOOL;
	SquareTimerDone : BOOL;
	StartBeltTimerDone : BOOL;
	TON_0 : TON;
	TON_1 : TON;
	TON_2 : TON;
	TON_3 : TON;
	TrailDelay1Done : BOOL;
	TON_4 : TON;
	LBPartSquared : BOOL;
	TON_5 : TON;
	LBBeamDownDone : BOOL;
	TON_6 : TON;
	EjectDwellDone : BOOL;
	LBWN12 : BOOL;
	MoveStarted : BOOL;
	TON_7 : TON;
	ReturnMoveStart : BOOL;
END_VAR
```

#### Cyclic.ld
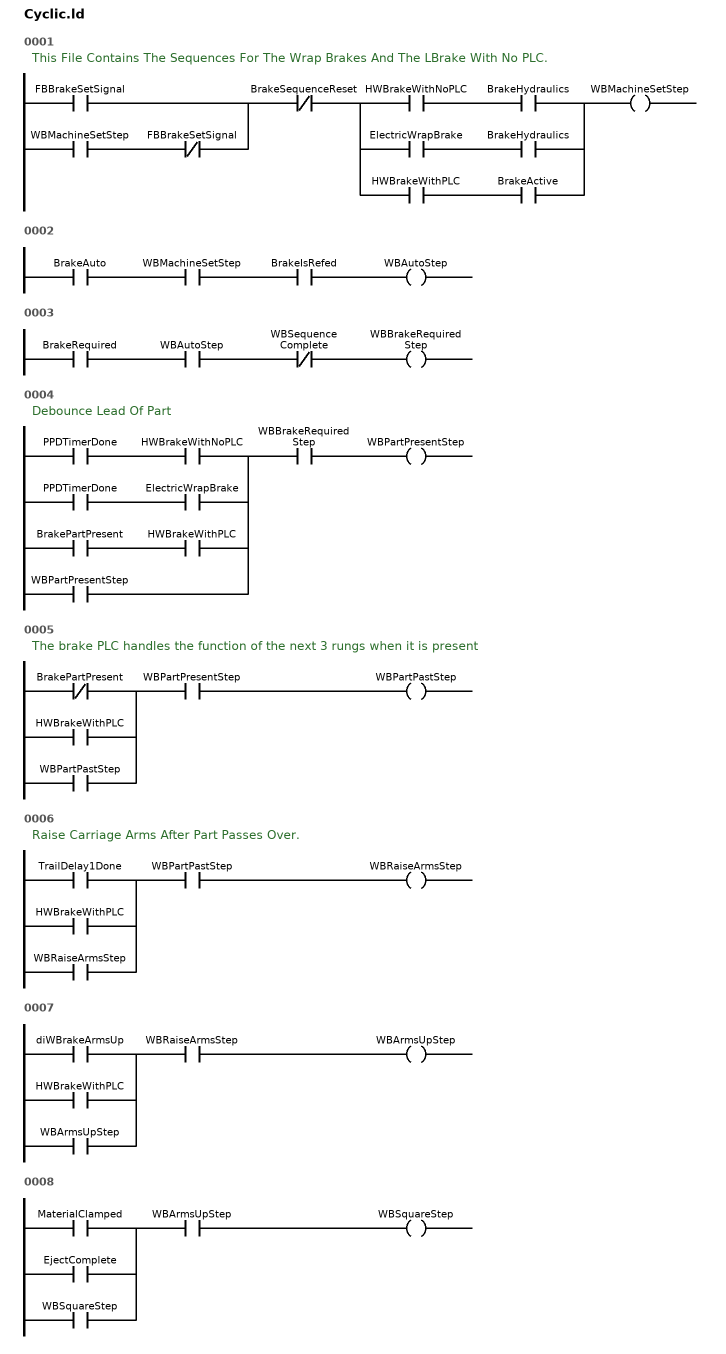
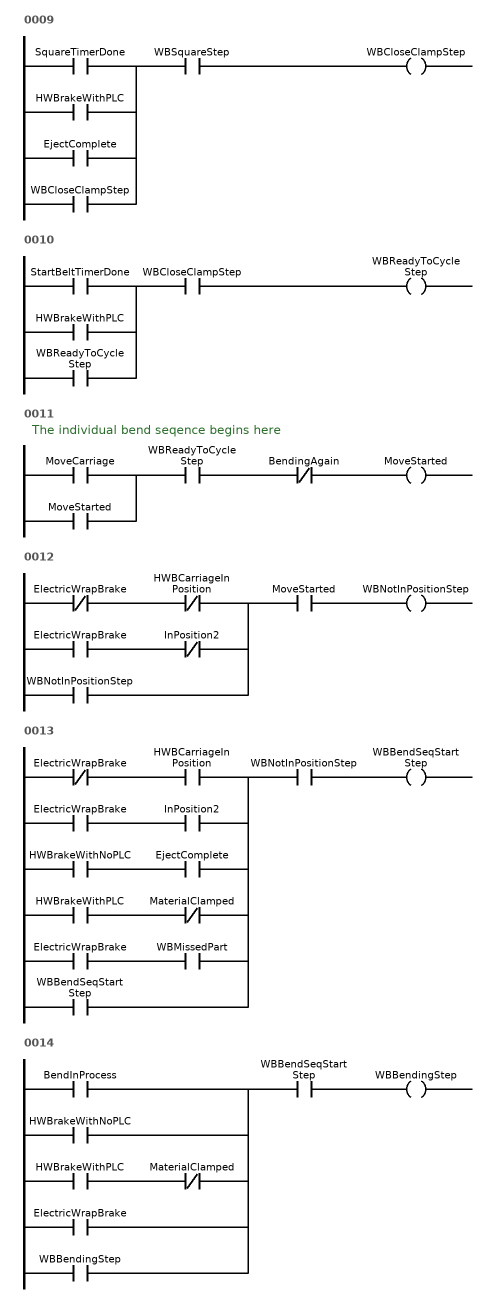
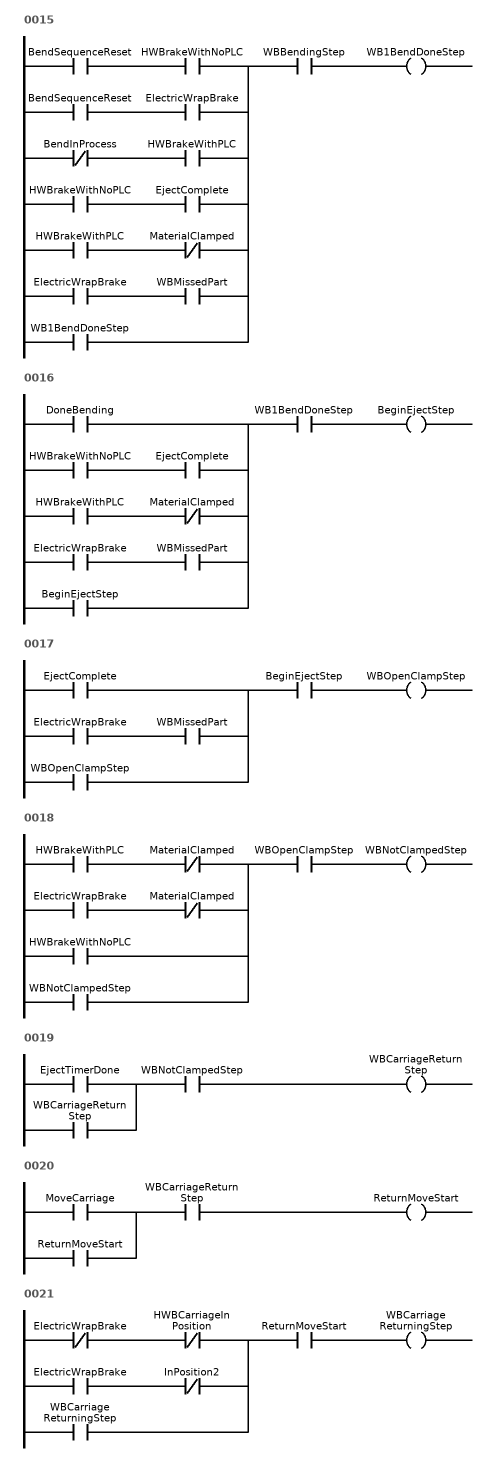
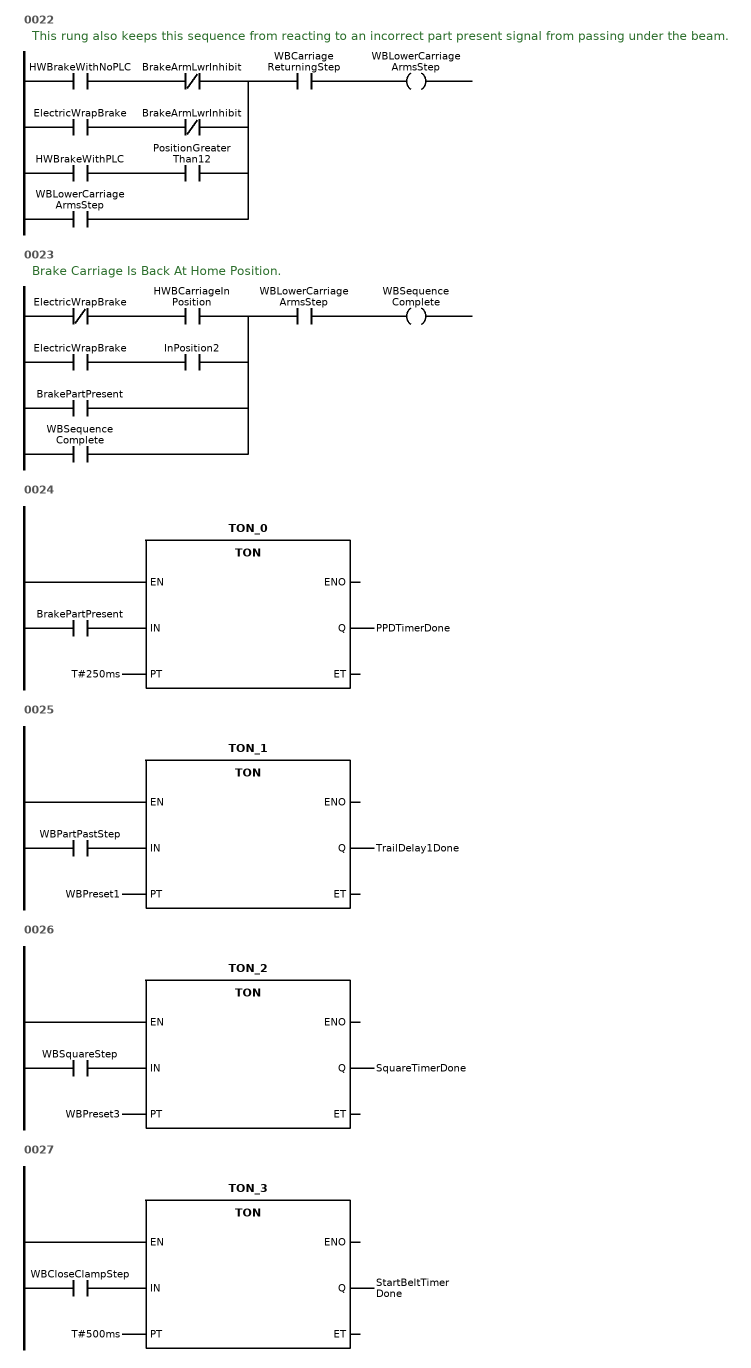
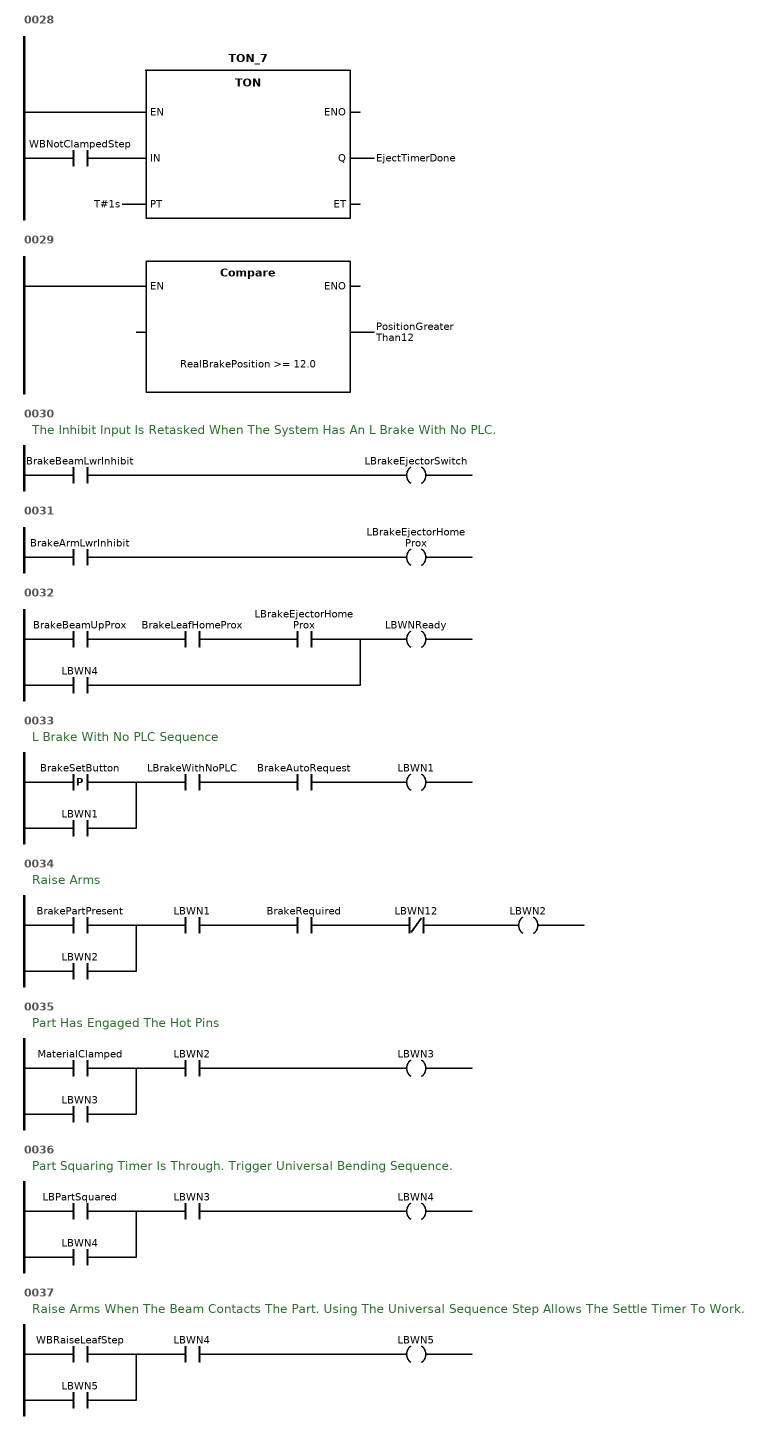
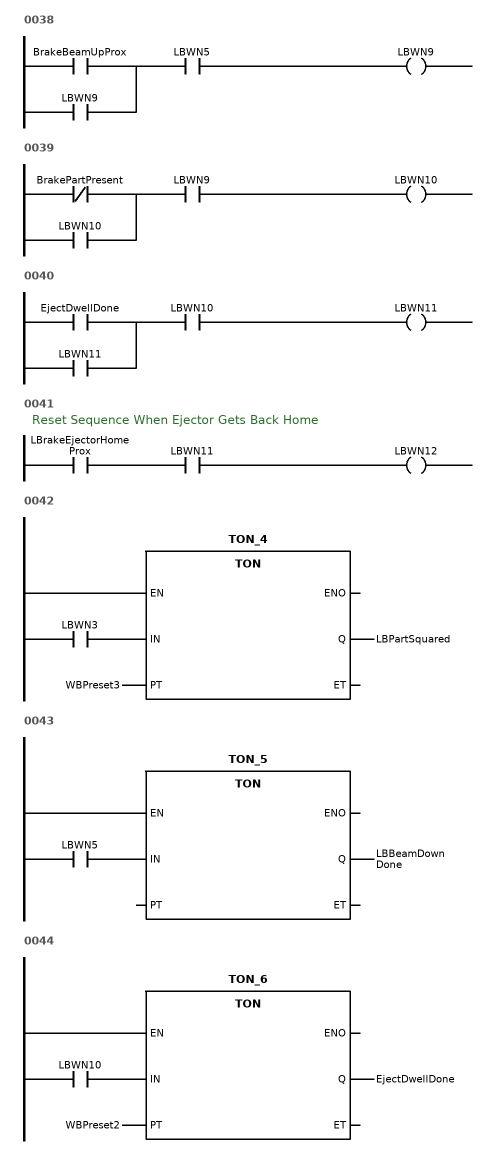
Ladder, written as Structured Text:
```iecst
PROGRAM _CYCLIC
VAR
    _p1 : BOOL;
    _e2 : R_TRIG;
END_VAR
(* Network 1: This File Contains The Sequences For The Wrap Brakes And The LBrake With No PLC. *)
_p1 := (FBBrakeSetSignal OR (WBMachineSetStep AND NOT FBBrakeSetSignal)) AND NOT BrakeSequenceReset;
WBMachineSetStep := _p1 AND ((HWBrakeWithNoPLC AND BrakeHydraulics) OR (ElectricWrapBrake AND BrakeHydraulics) OR (HWBrakeWithPLC AND BrakeActive));

(* Network 2 *)
WBAutoStep := BrakeAuto AND WBMachineSetStep AND BrakeIsRefed;

(* Network 3 *)
WBBrakeRequiredStep := BrakeRequired AND WBAutoStep AND NOT WBSequenceComplete;

(* Network 4: Debounce Lead Of Part *)
WBPartPresentStep := ((PPDTimerDone AND (HWBrakeWithNoPLC OR ElectricWrapBrake)) OR (BrakePartPresent AND HWBrakeWithPLC) OR WBPartPresentStep) AND WBBrakeRequiredStep;

(* Network 5: The brake PLC handles the function of the next 3 rungs when it is present *)
WBPartPastStep := (NOT BrakePartPresent OR HWBrakeWithPLC OR WBPartPastStep) AND WBPartPresentStep;

(* Network 6: Raise Carriage Arms After Part Passes Over. *)
WBRaiseArmsStep := (TrailDelay1Done OR HWBrakeWithPLC OR WBRaiseArmsStep) AND WBPartPastStep;

(* Network 7 *)
WBArmsUpStep := (diWBrakeArmsUp OR HWBrakeWithPLC OR WBArmsUpStep) AND WBRaiseArmsStep;

(* Network 8 *)
WBSquareStep := (MaterialClamped OR EjectComplete OR WBSquareStep) AND WBArmsUpStep;

(* Network 9 *)
WBCloseClampStep := (SquareTimerDone OR HWBrakeWithPLC OR EjectComplete OR WBCloseClampStep) AND WBSquareStep;

(* Network 10 *)
WBReadyToCycleStep := (StartBeltTimerDone OR HWBrakeWithPLC OR WBReadyToCycleStep) AND WBCloseClampStep;

(* Network 11: The individual bend seqence begins here *)
MoveStarted := (MoveCarriage OR MoveStarted) AND WBReadyToCycleStep AND NOT BendingAgain;

(* Network 12 *)
WBNotInPositionStep := ((NOT ElectricWrapBrake AND NOT HWBCarriageInPosition) OR (ElectricWrapBrake AND NOT InPosition2) OR WBNotInPositionStep) AND MoveStarted;

(* Network 13 *)
WBBendSeqStartStep := ((NOT ElectricWrapBrake AND HWBCarriageInPosition) OR (ElectricWrapBrake AND InPosition2) OR (HWBrakeWithNoPLC AND EjectComplete) OR (HWBrakeWithPLC AND NOT MaterialClamped) OR (ElectricWrapBrake AND WBMissedPart) OR WBBendSeqStartStep) AND WBNotInPositionStep;

(* Network 14 *)
WBBendingStep := (BendInProcess OR HWBrakeWithNoPLC OR (HWBrakeWithPLC AND NOT MaterialClamped) OR ElectricWrapBrake OR WBBendingStep) AND WBBendSeqStartStep;

(* Network 15 *)
WB1BendDoneStep := ((BendSequenceReset AND (HWBrakeWithNoPLC OR ElectricWrapBrake)) OR (NOT BendInProcess AND HWBrakeWithPLC) OR (HWBrakeWithNoPLC AND EjectComplete) OR (HWBrakeWithPLC AND NOT MaterialClamped) OR (ElectricWrapBrake AND WBMissedPart) OR WB1BendDoneStep) AND WBBendingStep;

(* Network 16 *)
BeginEjectStep := (DoneBending OR (HWBrakeWithNoPLC AND EjectComplete) OR (HWBrakeWithPLC AND NOT MaterialClamped) OR (ElectricWrapBrake AND WBMissedPart) OR BeginEjectStep) AND WB1BendDoneStep;

(* Network 17 *)
WBOpenClampStep := (EjectComplete OR (ElectricWrapBrake AND WBMissedPart) OR WBOpenClampStep) AND BeginEjectStep;

(* Network 18 *)
WBNotClampedStep := ((HWBrakeWithPLC AND NOT MaterialClamped) OR (ElectricWrapBrake AND NOT MaterialClamped) OR HWBrakeWithNoPLC OR WBNotClampedStep) AND WBOpenClampStep;

(* Network 19 *)
WBCarriageReturnStep := (EjectTimerDone OR WBCarriageReturnStep) AND WBNotClampedStep;

(* Network 20 *)
ReturnMoveStart := (MoveCarriage OR ReturnMoveStart) AND WBCarriageReturnStep;

(* Network 21 *)
WBCarriageReturningStep := ((NOT ElectricWrapBrake AND NOT HWBCarriageInPosition) OR (ElectricWrapBrake AND NOT InPosition2) OR WBCarriageReturningStep) AND ReturnMoveStart;

(* Network 22: This rung also keeps this sequence from reacting to an incorrect part present signal from passing under the beam. *)
WBLowerCarriageArmsStep := ((HWBrakeWithNoPLC AND NOT BrakeArmLwrInhibit) OR (ElectricWrapBrake AND NOT BrakeArmLwrInhibit) OR (HWBrakeWithPLC AND PositionGreaterThan12) OR WBLowerCarriageArmsStep) AND WBCarriageReturningStep;

(* Network 23: Brake Carriage Is Back At Home Position. *)
WBSequenceComplete := ((NOT ElectricWrapBrake AND HWBCarriageInPosition) OR (ElectricWrapBrake AND InPosition2) OR BrakePartPresent OR WBSequenceComplete) AND WBLowerCarriageArmsStep;

(* Network 24 *)
TON_0(IN := BrakePartPresent, PT := T#250ms);
PPDTimerDone := TON_0.Q;

(* Network 25 *)
TON_1(IN := WBPartPastStep, PT := WBPreset1);
TrailDelay1Done := TON_1.Q;

(* Network 26 *)
TON_2(IN := WBSquareStep, PT := WBPreset3);
SquareTimerDone := TON_2.Q;

(* Network 27 *)
TON_3(IN := WBCloseClampStep, PT := T#500ms);
StartBeltTimerDone := TON_3.Q;

(* Network 28 *)
TON_7(IN := WBNotClampedStep, PT := T#1s);
EjectTimerDone := TON_7.Q;

(* Network 29 *)
PositionGreaterThan12 := RealBrakePosition >= 12.0;

(* Network 30: The Inhibit Input Is Retasked When The System Has An L Brake With No PLC. *)
LBrakeEjectorSwitch := BrakeBeamLwrInhibit;

(* Network 31 *)
LBrakeEjectorHomeProx := BrakeArmLwrInhibit;

(* Network 32 *)
LBWNReady := (BrakeBeamUpProx AND BrakeLeafHomeProx AND LBrakeEjectorHomeProx) OR LBWN4;

(* Network 33: L Brake With No PLC Sequence *)
_e2(CLK := BrakeSetButton);
LBWN1 := (_e2.Q OR LBWN1) AND LBrakeWithNoPLC AND BrakeAutoRequest;

(* Network 34: Raise Arms *)
LBWN2 := (BrakePartPresent OR LBWN2) AND LBWN1 AND BrakeRequired AND NOT LBWN12;

(* Network 35: Part Has Engaged The Hot Pins *)
LBWN3 := (MaterialClamped OR LBWN3) AND LBWN2;

(* Network 36: Part Squaring Timer Is Through. Trigger Universal Bending Sequence. *)
LBWN4 := (LBPartSquared OR LBWN4) AND LBWN3;

(* Network 37: Raise Arms When The Beam Contacts The Part. Using The Universal Sequence Step Allows The Settle Timer To Work. *)
LBWN5 := (WBRaiseLeafStep OR LBWN5) AND LBWN4;

(* Network 38 *)
LBWN9 := (BrakeBeamUpProx OR LBWN9) AND LBWN5;

(* Network 39 *)
LBWN10 := (NOT BrakePartPresent OR LBWN10) AND LBWN9;

(* Network 40 *)
LBWN11 := (EjectDwellDone OR LBWN11) AND LBWN10;

(* Network 41: Reset Sequence When Ejector Gets Back Home *)
LBWN12 := LBrakeEjectorHomeProx AND LBWN11;

(* Network 42 *)
TON_4(IN := LBWN3, PT := WBPreset3);
LBPartSquared := TON_4.Q;

(* Network 43 *)
TON_5(IN := LBWN5);
LBBeamDownDone := TON_5.Q;

(* Network 44 *)
TON_6(IN := LBWN10, PT := WBPreset2);
EjectDwellDone := TON_6.Q;
END_PROGRAM
```

### Program Logical/TDCTable (IEC)

#### Variables.var
```iecst
VAR
	MarkSetComplete : BOOL;
	Cycle6 : BOOL;
	Cycle1 : BOOL;
	PartSquared : BOOL;
	Cycle2 : BOOL;
	Cycle3 : BOOL;
	PusherPaused : BOOL;
	Cycle4 : BOOL;
	Cycle5 : BOOL;
	DwellDone : BOOL;
	PartSettleDelay : TIME;
	TON_0 : TON;
	PauseDwell : TIME;
	TON_1 : TON;
	TDCPartLength : REAL;
	TableSpeed : REAL := 10.0;
	PusherDwellTime : TIME;
	UseMinDwell : BOOL;
	TON_2 : TON;
	TP_0 : TP;
	SetupPulse : BOOL;
	TON_3 : TON;
	KnurledRoll : BOOL;
	PushReverse : BOOL;
	PusherDwellReal : REAL;
	TP_1 : TP;
	DuctTypeEquals0 : BOOL;
END_VAR
```
